{attribute 'GeneratedUsingTerminal: EL1259-0000-0016'}
{attribute addProperty BoxType "EL1259-0000-0016"}
{attribute addProperty Id "CtrlAT %Q*Ctrl_B05F80DF5OutputsAT %Q*Outputs_A910484D10Output_event_timeAT %Q*ARRAY[0..9] OF UDINT40"}
{attribute addProperty CRC "2275852249"}
{attribute addProperty Size "55"}
TYPE MTO_Outputs_10x_Channel_232E0117 EXTENDS OutputBase_10CEE7DE :
STRUCT
	{attribute addProperty Name "Ctrl"}
	Ctrl AT %Q* : Ctrl_B05F80DF;
	{attribute addProperty Name "Outputs"}
	Outputs AT %Q* : Outputs_A910484D;
	{attribute addProperty Name "Output_event_time"}
	Output_event_time AT %Q* : ARRAY[0..9] OF UDINT;
END_STRUCT
END_TYPE

(* stored: Version 1.2.0.0, ProductVersion 3.1.4024.9
   DUT MTO_Outputs_10x_Channel_232E0117: Id {d7cc8d4a-31a5-4b55-b4cb-c45554aa0b2d} *)
